FUNCTION F_UpdateTimeWithSystemTime
VAR_INPUT
	stEvent : REFERENCE TO ST_Event;
END_VAR
VAR
	fbGETSYSTEMTIME : GETSYSTEMTIME;
	stFileTime : T_FILETIME;
END_VAR

fbGETSYSTEMTIME(timeLoDW => stFileTime.dwLowDateTime,
				timeHiDW => stFileTime.dwHighDateTime);
stEvent.dtTimestamp := FILETIME_TO_DT(fileTime := stFileTime);

END_FUNCTION

(* stored: Version 1.1.0.1, ProductVersion 3.1.4024.16
   POU F_UpdateTimeWithSystemTime: Id {d547d8c5-553d-4f86-ab92-3bd997f19374}, SpecialFunc None *)
